PROGRAM MAIN
VAR
	ESTACION: FB_Estacion;
END_VAR

IF NOT ESTACION.SelectorManual THEN
	ESTACION();
END_IF

END_PROGRAM

(* stored: Version 1.1.0.1, ProductVersion 3.1.4024.12
   POU MAIN: Id {2f866281-c418-478f-8ac3-95bfd1520d77}, SpecialFunc None *)
